FUNCTION_BLOCK BOOLS_TO_QUARTERS (* Composite FB wrapping other FBs *)
  (* Standard: 61499-2; Description: Copyright (c) 2024 HR Agrartechnik GmbH This program and the accompanying materials are made available under the terms of the Eclipse Public License 2.0 which is available at https://www.eclipse.org/legal/epl-2.0/ SPDX-License-Identifier: EPL-2.0 *)
  (* Version 1.0, 2024-02-29, Franz Höpfinger, HR Agrartechnik GmbH *)
  PACKAGE logiBUS::utils::quarter;
  IMPORT logiBUS::utils::quarter::const::quarter;
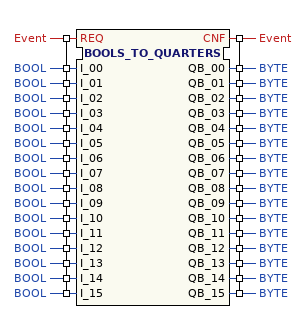
  EVENT_INPUT
    REQ WITH I_00, I_01, I_02, I_03, I_04, I_05, I_06, I_07, I_08, I_09, I_10, I_11, I_12, I_13, I_14, I_15; (* Normal Execution Request *)
  END_EVENT
  EVENT_OUTPUT
    CNF WITH QB_00, QB_01, QB_02, QB_03, QB_04, QB_05, QB_06, QB_07, QB_08, QB_09, QB_10, QB_11, QB_12, QB_13, QB_14, QB_15; (* Execution Confirmation *)
  END_EVENT
  VAR_INPUT
    I_00 : BOOL := BOOL#FALSE; (* BOOL Input *)
    I_01 : BOOL := BOOL#FALSE; (* BOOL Input *)
    I_02 : BOOL := BOOL#FALSE; (* BOOL Input *)
    I_03 : BOOL := BOOL#FALSE; (* BOOL Input *)
    I_04 : BOOL := BOOL#FALSE; (* BOOL Input *)
    I_05 : BOOL := BOOL#FALSE; (* BOOL Input *)
    I_06 : BOOL := BOOL#FALSE; (* BOOL Input *)
    I_07 : BOOL := BOOL#FALSE; (* BOOL Input *)
    I_08 : BOOL := BOOL#FALSE; (* BOOL Input *)
    I_09 : BOOL := BOOL#FALSE; (* BOOL Input *)
    I_10 : BOOL := BOOL#FALSE; (* BOOL Input *)
    I_11 : BOOL := BOOL#FALSE; (* BOOL Input *)
    I_12 : BOOL := BOOL#FALSE; (* BOOL Input *)
    I_13 : BOOL := BOOL#FALSE; (* BOOL Input *)
    I_14 : BOOL := BOOL#FALSE; (* BOOL Input *)
    I_15 : BOOL := BOOL#FALSE; (* BOOL Input *)
  END_VAR
  VAR_OUTPUT
    QB_00 : BYTE := quarter::COMMAND_DISABLE; (* 2bit (quarter Byte) Output with 4 States (only 2 used) *)
    QB_01 : BYTE := quarter::COMMAND_DISABLE; (* 2bit (quarter Byte) Output with 4 States (only 2 used) *)
    QB_02 : BYTE := quarter::COMMAND_DISABLE; (* 2bit (quarter Byte) Output with 4 States (only 2 used) *)
    QB_03 : BYTE := quarter::COMMAND_DISABLE; (* 2bit (quarter Byte) Output with 4 States (only 2 used) *)
    QB_04 : BYTE := quarter::COMMAND_DISABLE; (* 2bit (quarter Byte) Output with 4 States (only 2 used) *)
    QB_05 : BYTE := quarter::COMMAND_DISABLE; (* 2bit (quarter Byte) Output with 4 States (only 2 used) *)
    QB_06 : BYTE := quarter::COMMAND_DISABLE; (* 2bit (quarter Byte) Output with 4 States (only 2 used) *)
    QB_07 : BYTE := quarter::COMMAND_DISABLE; (* 2bit (quarter Byte) Output with 4 States (only 2 used) *)
    QB_08 : BYTE := quarter::COMMAND_DISABLE; (* 2bit (quarter Byte) Output with 4 States (only 2 used) *)
    QB_09 : BYTE := quarter::COMMAND_DISABLE; (* 2bit (quarter Byte) Output with 4 States (only 2 used) *)
    QB_10 : BYTE := quarter::COMMAND_DISABLE; (* 2bit (quarter Byte) Output with 4 States (only 2 used) *)
    QB_11 : BYTE := quarter::COMMAND_DISABLE; (* 2bit (quarter Byte) Output with 4 States (only 2 used) *)
    QB_12 : BYTE := quarter::COMMAND_DISABLE; (* 2bit (quarter Byte) Output with 4 States (only 2 used) *)
    QB_13 : BYTE := quarter::COMMAND_DISABLE; (* 2bit (quarter Byte) Output with 4 States (only 2 used) *)
    QB_14 : BYTE := quarter::COMMAND_DISABLE; (* 2bit (quarter Byte) Output with 4 States (only 2 used) *)
    QB_15 : BYTE := quarter::COMMAND_DISABLE; (* 2bit (quarter Byte) Output with 4 States (only 2 used) *)
  END_VAR
  FBS
    BOOL_TO_QUARTER_00 : logiBUS::utils::quarter::BOOL_TO_QUARTER;
    BOOL_TO_QUARTER_01 : logiBUS::utils::quarter::BOOL_TO_QUARTER;
    BOOL_TO_QUARTER_02 : logiBUS::utils::quarter::BOOL_TO_QUARTER;
    BOOL_TO_QUARTER_03 : logiBUS::utils::quarter::BOOL_TO_QUARTER;
    BOOL_TO_QUARTER_04 : logiBUS::utils::quarter::BOOL_TO_QUARTER;
    BOOL_TO_QUARTER_05 : logiBUS::utils::quarter::BOOL_TO_QUARTER;
    BOOL_TO_QUARTER_06 : logiBUS::utils::quarter::BOOL_TO_QUARTER;
    BOOL_TO_QUARTER_07 : logiBUS::utils::quarter::BOOL_TO_QUARTER;
    BOOL_TO_QUARTER_08 : logiBUS::utils::quarter::BOOL_TO_QUARTER;
    BOOL_TO_QUARTER_09 : logiBUS::utils::quarter::BOOL_TO_QUARTER;
    BOOL_TO_QUARTER_10 : logiBUS::utils::quarter::BOOL_TO_QUARTER;
    BOOL_TO_QUARTER_11 : logiBUS::utils::quarter::BOOL_TO_QUARTER;
    BOOL_TO_QUARTER_12 : logiBUS::utils::quarter::BOOL_TO_QUARTER;
    BOOL_TO_QUARTER_13 : logiBUS::utils::quarter::BOOL_TO_QUARTER;
    BOOL_TO_QUARTER_14 : logiBUS::utils::quarter::BOOL_TO_QUARTER;
    BOOL_TO_QUARTER_15 : logiBUS::utils::quarter::BOOL_TO_QUARTER;
  END_FBS
  EVENT_CONNECTIONS
    REQ TO BOOL_TO_QUARTER_00.REQ;
    BOOL_TO_QUARTER_00.CNF TO BOOL_TO_QUARTER_01.REQ;
    BOOL_TO_QUARTER_01.CNF TO BOOL_TO_QUARTER_02.REQ;
    BOOL_TO_QUARTER_02.CNF TO BOOL_TO_QUARTER_03.REQ;
    BOOL_TO_QUARTER_03.CNF TO BOOL_TO_QUARTER_04.REQ;
    BOOL_TO_QUARTER_04.CNF TO BOOL_TO_QUARTER_05.REQ;
    BOOL_TO_QUARTER_05.CNF TO BOOL_TO_QUARTER_06.REQ;
    BOOL_TO_QUARTER_06.CNF TO BOOL_TO_QUARTER_07.REQ;
    BOOL_TO_QUARTER_07.CNF TO BOOL_TO_QUARTER_08.REQ;
    BOOL_TO_QUARTER_08.CNF TO BOOL_TO_QUARTER_09.REQ;
    BOOL_TO_QUARTER_09.CNF TO BOOL_TO_QUARTER_10.REQ;
    BOOL_TO_QUARTER_10.CNF TO BOOL_TO_QUARTER_11.REQ;
    BOOL_TO_QUARTER_11.CNF TO BOOL_TO_QUARTER_12.REQ;
    BOOL_TO_QUARTER_12.CNF TO BOOL_TO_QUARTER_13.REQ;
    BOOL_TO_QUARTER_13.CNF TO BOOL_TO_QUARTER_14.REQ;
    BOOL_TO_QUARTER_14.CNF TO BOOL_TO_QUARTER_15.REQ;
    BOOL_TO_QUARTER_15.CNF TO CNF;
  END_CONNECTIONS
  DATA_CONNECTIONS
    I_00 TO BOOL_TO_QUARTER_00.I;
    BOOL_TO_QUARTER_00. TO QB_00;
    I_01 TO BOOL_TO_QUARTER_01.I;
    BOOL_TO_QUARTER_01. TO QB_01;
    I_02 TO BOOL_TO_QUARTER_02.I;
    BOOL_TO_QUARTER_02. TO QB_02;
    I_03 TO BOOL_TO_QUARTER_03.I;
    I_04 TO BOOL_TO_QUARTER_04.I;
    BOOL_TO_QUARTER_05. TO QB_05;
    BOOL_TO_QUARTER_04. TO QB_04;
    BOOL_TO_QUARTER_03. TO QB_03;
    I_06 TO BOOL_TO_QUARTER_06.I;
    BOOL_TO_QUARTER_06. TO QB_06;
    BOOL_TO_QUARTER_15. TO QB_15;
    BOOL_TO_QUARTER_07. TO QB_07;
    BOOL_TO_QUARTER_08. TO QB_08;
    BOOL_TO_QUARTER_09. TO QB_09;
    BOOL_TO_QUARTER_10. TO QB_10;
    BOOL_TO_QUARTER_11. TO QB_11;
    BOOL_TO_QUARTER_12. TO QB_12;
    BOOL_TO_QUARTER_13. TO QB_13;
    BOOL_TO_QUARTER_14. TO QB_14;
    I_05 TO BOOL_TO_QUARTER_05.I;
    I_07 TO BOOL_TO_QUARTER_07.I;
    I_08 TO BOOL_TO_QUARTER_08.I;
    I_09 TO BOOL_TO_QUARTER_09.I;
    I_10 TO BOOL_TO_QUARTER_10.I;
    I_11 TO BOOL_TO_QUARTER_11.I;
    I_12 TO BOOL_TO_QUARTER_12.I;
    I_13 TO BOOL_TO_QUARTER_13.I;
    I_14 TO BOOL_TO_QUARTER_14.I;
    I_15 TO BOOL_TO_QUARTER_15.I;
  END_CONNECTIONS
END_FUNCTION_BLOCK
